ABB RAPID module: Calib_mg_test_230111.modx

MODULE Calib_mg_test_230111(READONLY)
 LOCAL CONST string dataName := "mg_test_230111";
 LOCAL CONST string mechUnitRef := "ROB_1";
 LOCAL CONST string toolRef := "tool0";
 LOCAL CONST robtarget pTCP_Point1 := [[247.2003,50.78513,455.9486],[0.5185382,-0.08632798,0.8490512,0.05270384],[0,-1,-1,0],[8.999999E+09,8.999999E+09,8.999999E+09,8.999999E+09,8.999999E+09,8.999999E+09]];
 LOCAL CONST robtarget pTCP_Point2 := [[267.8177,50.7888,455.9514],[0.2497867,-0.06756534,0.9659405,-0.0007212608],[0,-1,0,0],[8.999999E+09,8.999999E+09,8.999999E+09,8.999999E+09,8.999999E+09,8.999999E+09]];
 LOCAL CONST robtarget pTCP_Point3 := [[267.8267,50.79159,455.9572],[0.05526131,0.02307686,0.9831463,-0.1727338],[0,-1,0,0],[8.999999E+09,8.999999E+09,8.999999E+09,8.999999E+09,8.999999E+09,8.999999E+09]];
 !------------------------------------------------------------------------------
 !<auto-generated>
 !This code was generated by a tool.

 !<auto-generated>
 !Changes to this file may cause incorrect behavior and will be lost if
 !the code is regenerated.
 !</auto-generated>
 !------------------------------------------------------------------------------



 ! 11 Jan 2023 11:12:44 by Default User from ABB Robotics FlexPendant
 ! Old Value: [TRUE,[[0,0,0],[1,0,0,0]],[0.2,[0,0,0],[1,0,0,0],0,0,0]]
 ! Maxerror, Minerror, Meanerror Values: 3.803636, 3.803636, 3.803636


ENDMODULE
